FUNCTION proj12_TupleStruct_1: LREAL
{ S7_Optimized_Access := 'true' }
    VAR_INPUT
        tuple: TupleStruct_1;
    END_VAR

BEGIN
    proj12_TupleStruct_1 := tuple.field12;
END_FUNCTION
